// Mitsubishi GX Works2 project: v05-1   PLC: Q02/Q02H

PROGRAM MAIN
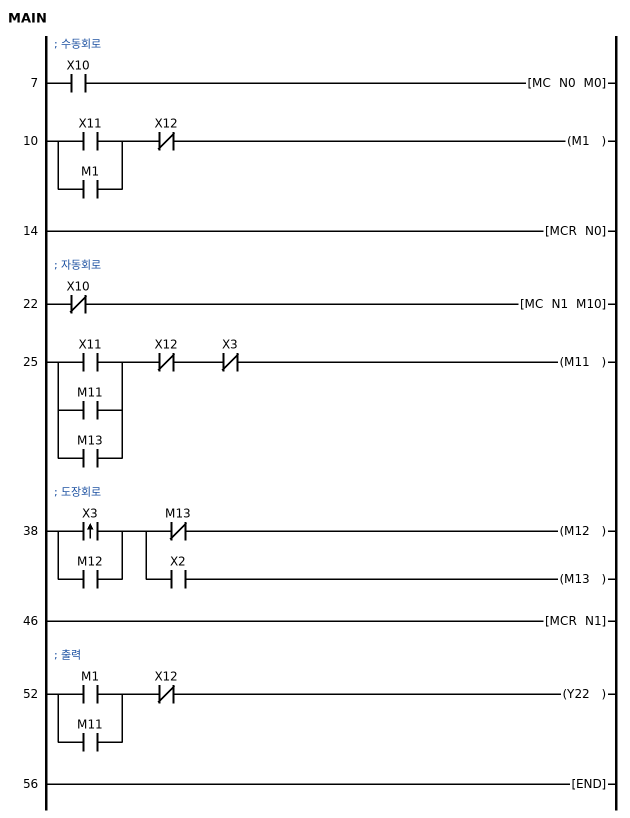
; 수동회로
7     LD      X10
      MC      N0 M0
10    LD      X11
      OR      M1
      ANI     X12
      OUT     M1
14    MCR     N0
; 자동회로
22    LDI     X10
      MC      N1 M10
25    LD      X11
      OR      M11
      OR      M13
      ANI     X12
      ANI     X3
      OUT     M11
; 도장회로
38    LDP     X3
      OR      M12
      MPS
      ANI     M13
      OUT     M12
      MPP
      AND     X2
      OUT     M13
46    MCR     N1
; 출력
52    LD      M1
      OR      M11
      ANI     X12
      OUT     Y22
56    END
END_PROGRAM
